TYPE "Decoiler_Status"
VERSION : 0.1
// Block: Decoiler_Status
   STRUCT
      Feed : SpeedMachine_COut;
      Jaws : ValveMachine_COut;
      Coupling : ValveMachine_COut;
      SnubberLift : ValveMachine_COut;
      SnubberRoll : ValveMachine_COut;
      CoilDiameter : Real;
      EndOfCoil : Bool;
      CouplingEngaged : Bool;
   END_STRUCT;

END_TYPE
